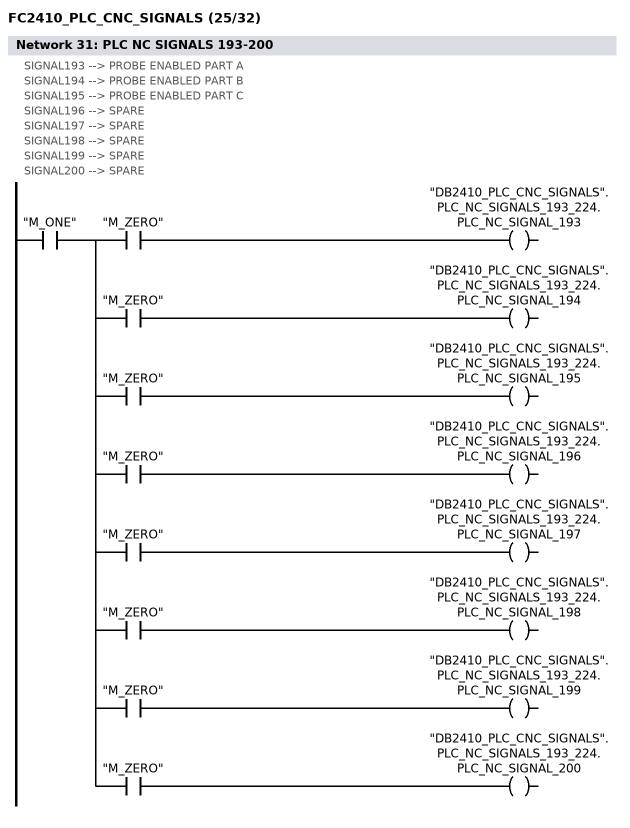
   RUNG wire#powerrail
      Contact( "M_ONE" )
      wire#w1
      Contact( "M_ZERO" )
      Coil( "DB2410_PLC_CNC_SIGNALS".PLC_NC_SIGNALS_193_224.PLC_NC_SIGNAL_193 )
   END_RUNG
   RUNG wire#w1
      Contact( "M_ZERO" )
      Coil( "DB2410_PLC_CNC_SIGNALS".PLC_NC_SIGNALS_193_224.PLC_NC_SIGNAL_194 )
   END_RUNG
   RUNG wire#w1
      Contact( "M_ZERO" )
      Coil( "DB2410_PLC_CNC_SIGNALS".PLC_NC_SIGNALS_193_224.PLC_NC_SIGNAL_195 )
   END_RUNG
   RUNG wire#w1
      Contact( "M_ZERO" )
      Coil( "DB2410_PLC_CNC_SIGNALS".PLC_NC_SIGNALS_193_224.PLC_NC_SIGNAL_196 )
   END_RUNG
   RUNG wire#w1
      Contact( "M_ZERO" )
      Coil( "DB2410_PLC_CNC_SIGNALS".PLC_NC_SIGNALS_193_224.PLC_NC_SIGNAL_197 )
   END_RUNG
   RUNG wire#w1
      Contact( "M_ZERO" )
      Coil( "DB2410_PLC_CNC_SIGNALS".PLC_NC_SIGNALS_193_224.PLC_NC_SIGNAL_198 )
   END_RUNG
   RUNG wire#w1
      Contact( "M_ZERO" )
      Coil( "DB2410_PLC_CNC_SIGNALS".PLC_NC_SIGNALS_193_224.PLC_NC_SIGNAL_199 )
   END_RUNG
   RUNG wire#w1
      Contact( "M_ZERO" )
      Coil( "DB2410_PLC_CNC_SIGNALS".PLC_NC_SIGNALS_193_224.PLC_NC_SIGNAL_200 )
   END_RUNG
   // the same network as SCL:
   "DB2410_PLC_CNC_SIGNALS".PLC_NC_SIGNALS_193_224.PLC_NC_SIGNAL_193 := "M_ONE" AND "M_ZERO";
   "DB2410_PLC_CNC_SIGNALS".PLC_NC_SIGNALS_193_224.PLC_NC_SIGNAL_194 := "M_ONE" AND "M_ZERO";
   "DB2410_PLC_CNC_SIGNALS".PLC_NC_SIGNALS_193_224.PLC_NC_SIGNAL_195 := "M_ONE" AND "M_ZERO";
   "DB2410_PLC_CNC_SIGNALS".PLC_NC_SIGNALS_193_224.PLC_NC_SIGNAL_196 := "M_ONE" AND "M_ZERO";
   "DB2410_PLC_CNC_SIGNALS".PLC_NC_SIGNALS_193_224.PLC_NC_SIGNAL_197 := "M_ONE" AND "M_ZERO";
   "DB2410_PLC_CNC_SIGNALS".PLC_NC_SIGNALS_193_224.PLC_NC_SIGNAL_198 := "M_ONE" AND "M_ZERO";
   "DB2410_PLC_CNC_SIGNALS".PLC_NC_SIGNALS_193_224.PLC_NC_SIGNAL_199 := "M_ONE" AND "M_ZERO";
   "DB2410_PLC_CNC_SIGNALS".PLC_NC_SIGNALS_193_224.PLC_NC_SIGNAL_200 := "M_ONE" AND "M_ZERO";
END_REGION

REGION Network 32: PLC NC SIGNALS 201-208
   // SIGNAL201 --> SPARE
   // SIGNAL202 --> SPARE
   // SIGNAL203 --> SPARE
   // SIGNAL204 --> SPARE
   // SIGNAL205 --> SPARE
   // SIGNAL206 --> SPARE
   // SIGNAL207 --> SPARE
   // SIGNAL208 --> SPARE
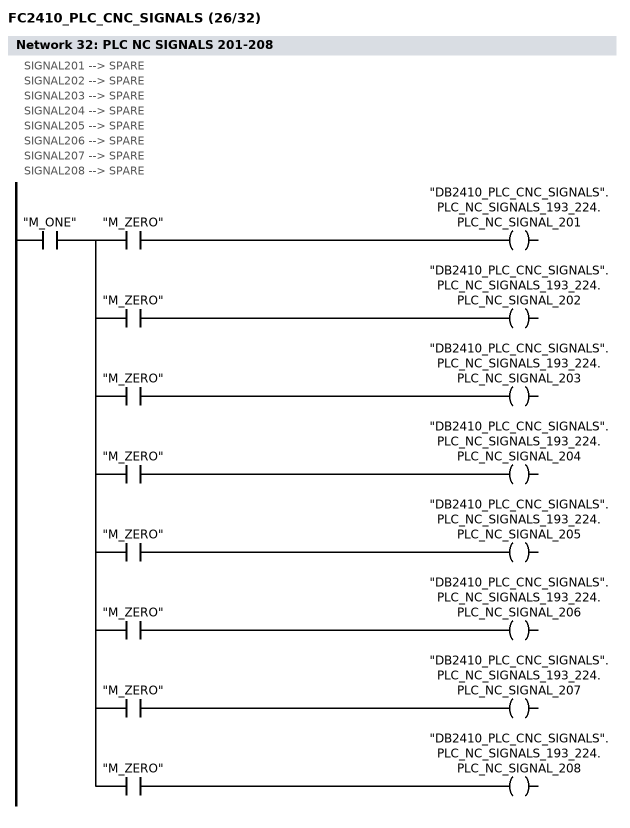
   RUNG wire#powerrail
      Contact( "M_ONE" )
      wire#w1
      Contact( "M_ZERO" )
      Coil( "DB2410_PLC_CNC_SIGNALS".PLC_NC_SIGNALS_193_224.PLC_NC_SIGNAL_201 )
   END_RUNG
   RUNG wire#w1
      Contact( "M_ZERO" )
      Coil( "DB2410_PLC_CNC_SIGNALS".PLC_NC_SIGNALS_193_224.PLC_NC_SIGNAL_202 )
   END_RUNG
   RUNG wire#w1
      Contact( "M_ZERO" )
      Coil( "DB2410_PLC_CNC_SIGNALS".PLC_NC_SIGNALS_193_224.PLC_NC_SIGNAL_203 )
   END_RUNG
   RUNG wire#w1
      Contact( "M_ZERO" )
      Coil( "DB2410_PLC_CNC_SIGNALS".PLC_NC_SIGNALS_193_224.PLC_NC_SIGNAL_204 )
   END_RUNG
   RUNG wire#w1
      Contact( "M_ZERO" )
      Coil( "DB2410_PLC_CNC_SIGNALS".PLC_NC_SIGNALS_193_224.PLC_NC_SIGNAL_205 )
   END_RUNG
   RUNG wire#w1
      Contact( "M_ZERO" )
      Coil( "DB2410_PLC_CNC_SIGNALS".PLC_NC_SIGNALS_193_224.PLC_NC_SIGNAL_206 )
   END_RUNG
   RUNG wire#w1
      Contact( "M_ZERO" )
      Coil( "DB2410_PLC_CNC_SIGNALS".PLC_NC_SIGNALS_193_224.PLC_NC_SIGNAL_207 )
   END_RUNG
   RUNG wire#w1
      Contact( "M_ZERO" )
      Coil( "DB2410_PLC_CNC_SIGNALS".PLC_NC_SIGNALS_193_224.PLC_NC_SIGNAL_208 )
   END_RUNG
   // the same network as SCL:
   "DB2410_PLC_CNC_SIGNALS".PLC_NC_SIGNALS_193_224.PLC_NC_SIGNAL_201 := "M_ONE" AND "M_ZERO";
   "DB2410_PLC_CNC_SIGNALS".PLC_NC_SIGNALS_193_224.PLC_NC_SIGNAL_202 := "M_ONE" AND "M_ZERO";
   "DB2410_PLC_CNC_SIGNALS".PLC_NC_SIGNALS_193_224.PLC_NC_SIGNAL_203 := "M_ONE" AND "M_ZERO";
   "DB2410_PLC_CNC_SIGNALS".PLC_NC_SIGNALS_193_224.PLC_NC_SIGNAL_204 := "M_ONE" AND "M_ZERO";
   "DB2410_PLC_CNC_SIGNALS".PLC_NC_SIGNALS_193_224.PLC_NC_SIGNAL_205 := "M_ONE" AND "M_ZERO";
   "DB2410_PLC_CNC_SIGNALS".PLC_NC_SIGNALS_193_224.PLC_NC_SIGNAL_206 := "M_ONE" AND "M_ZERO";
   "DB2410_PLC_CNC_SIGNALS".PLC_NC_SIGNALS_193_224.PLC_NC_SIGNAL_207 := "M_ONE" AND "M_ZERO";
   "DB2410_PLC_CNC_SIGNALS".PLC_NC_SIGNALS_193_224.PLC_NC_SIGNAL_208 := "M_ONE" AND "M_ZERO";
END_REGION

REGION Network 33: PLC NC SIGNALS 209-216
   // SIGNAL209 --> SPARE
   // SIGNAL210 --> SPARE
   // SIGNAL211 --> SPARE
   // SIGNAL212 --> SPARE
   // SIGNAL213 --> SPARE
   // SIGNAL214 --> SPARE
   // SIGNAL215 --> SPARE
   // SIGNAL216 --> SPARE
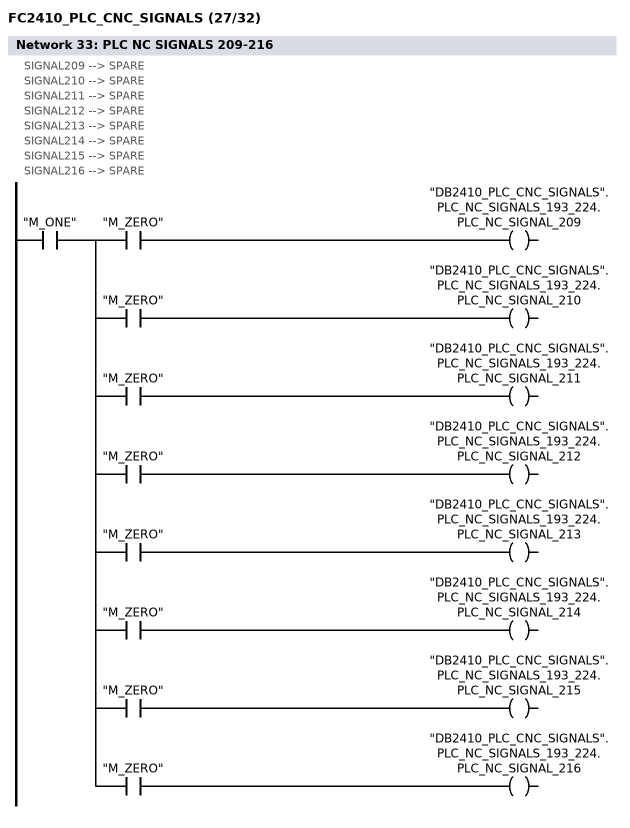
   RUNG wire#powerrail
      Contact( "M_ONE" )
      wire#w1
      Contact( "M_ZERO" )
      Coil( "DB2410_PLC_CNC_SIGNALS".PLC_NC_SIGNALS_193_224.PLC_NC_SIGNAL_209 )
   END_RUNG
   RUNG wire#w1
      Contact( "M_ZERO" )
      Coil( "DB2410_PLC_CNC_SIGNALS".PLC_NC_SIGNALS_193_224.PLC_NC_SIGNAL_210 )
   END_RUNG
   RUNG wire#w1
      Contact( "M_ZERO" )
      Coil( "DB2410_PLC_CNC_SIGNALS".PLC_NC_SIGNALS_193_224.PLC_NC_SIGNAL_211 )
   END_RUNG
   RUNG wire#w1
      Contact( "M_ZERO" )
      Coil( "DB2410_PLC_CNC_SIGNALS".PLC_NC_SIGNALS_193_224.PLC_NC_SIGNAL_212 )
   END_RUNG
   RUNG wire#w1
      Contact( "M_ZERO" )
      Coil( "DB2410_PLC_CNC_SIGNALS".PLC_NC_SIGNALS_193_224.PLC_NC_SIGNAL_213 )
   END_RUNG
   RUNG wire#w1
      Contact( "M_ZERO" )
      Coil( "DB2410_PLC_CNC_SIGNALS".PLC_NC_SIGNALS_193_224.PLC_NC_SIGNAL_214 )
   END_RUNG
   RUNG wire#w1
      Contact( "M_ZERO" )
      Coil( "DB2410_PLC_CNC_SIGNALS".PLC_NC_SIGNALS_193_224.PLC_NC_SIGNAL_215 )
   END_RUNG
   RUNG wire#w1
      Contact( "M_ZERO" )
      Coil( "DB2410_PLC_CNC_SIGNALS".PLC_NC_SIGNALS_193_224.PLC_NC_SIGNAL_216 )
   END_RUNG
   // the same network as SCL:
   "DB2410_PLC_CNC_SIGNALS".PLC_NC_SIGNALS_193_224.PLC_NC_SIGNAL_209 := "M_ONE" AND "M_ZERO";
   "DB2410_PLC_CNC_SIGNALS".PLC_NC_SIGNALS_193_224.PLC_NC_SIGNAL_210 := "M_ONE" AND "M_ZERO";
   "DB2410_PLC_CNC_SIGNALS".PLC_NC_SIGNALS_193_224.PLC_NC_SIGNAL_211 := "M_ONE" AND "M_ZERO";
   "DB2410_PLC_CNC_SIGNALS".PLC_NC_SIGNALS_193_224.PLC_NC_SIGNAL_212 := "M_ONE" AND "M_ZERO";
   "DB2410_PLC_CNC_SIGNALS".PLC_NC_SIGNALS_193_224.PLC_NC_SIGNAL_213 := "M_ONE" AND "M_ZERO";
   "DB2410_PLC_CNC_SIGNALS".PLC_NC_SIGNALS_193_224.PLC_NC_SIGNAL_214 := "M_ONE" AND "M_ZERO";
   "DB2410_PLC_CNC_SIGNALS".PLC_NC_SIGNALS_193_224.PLC_NC_SIGNAL_215 := "M_ONE" AND "M_ZERO";
   "DB2410_PLC_CNC_SIGNALS".PLC_NC_SIGNALS_193_224.PLC_NC_SIGNAL_216 := "M_ONE" AND "M_ZERO";
END_REGION

REGION Network 34: PLC NC SIGNALS 217-224
   // SIGNAL217 --> SPARE
   // SIGNAL218 --> SPARE
   // SIGNAL219 --> SPARE
   // SIGNAL220 --> SPARE
   // SIGNAL221 --> SPARE
   // SIGNAL222 --> SPARE
   // SIGNAL223 --> SPARE
   // SIGNAL224 --> SPARE
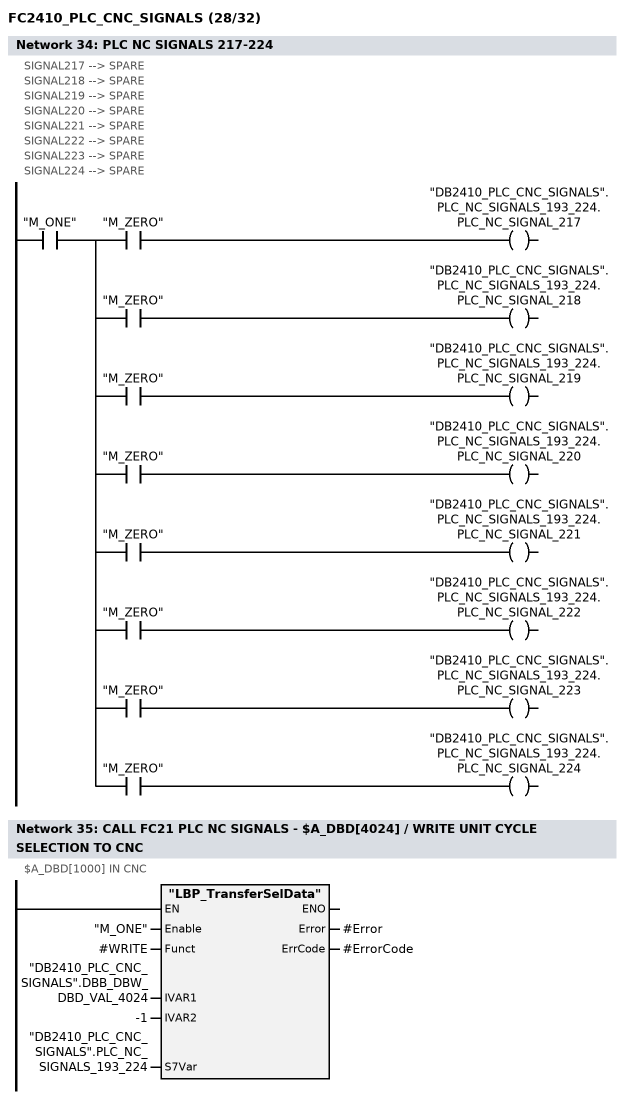
   RUNG wire#powerrail
      Contact( "M_ONE" )
      wire#w1
      Contact( "M_ZERO" )
      Coil( "DB2410_PLC_CNC_SIGNALS".PLC_NC_SIGNALS_193_224.PLC_NC_SIGNAL_217 )
   END_RUNG
   RUNG wire#w1
      Contact( "M_ZERO" )
      Coil( "DB2410_PLC_CNC_SIGNALS".PLC_NC_SIGNALS_193_224.PLC_NC_SIGNAL_218 )
   END_RUNG
   RUNG wire#w1
      Contact( "M_ZERO" )
      Coil( "DB2410_PLC_CNC_SIGNALS".PLC_NC_SIGNALS_193_224.PLC_NC_SIGNAL_219 )
   END_RUNG
   RUNG wire#w1
      Contact( "M_ZERO" )
      Coil( "DB2410_PLC_CNC_SIGNALS".PLC_NC_SIGNALS_193_224.PLC_NC_SIGNAL_220 )
   END_RUNG
   RUNG wire#w1
      Contact( "M_ZERO" )
      Coil( "DB2410_PLC_CNC_SIGNALS".PLC_NC_SIGNALS_193_224.PLC_NC_SIGNAL_221 )
   END_RUNG
   RUNG wire#w1
      Contact( "M_ZERO" )
      Coil( "DB2410_PLC_CNC_SIGNALS".PLC_NC_SIGNALS_193_224.PLC_NC_SIGNAL_222 )
   END_RUNG
   RUNG wire#w1
      Contact( "M_ZERO" )
      Coil( "DB2410_PLC_CNC_SIGNALS".PLC_NC_SIGNALS_193_224.PLC_NC_SIGNAL_223 )
   END_RUNG
   RUNG wire#w1
      Contact( "M_ZERO" )
      Coil( "DB2410_PLC_CNC_SIGNALS".PLC_NC_SIGNALS_193_224.PLC_NC_SIGNAL_224 )
   END_RUNG
   // the same network as SCL:
   "DB2410_PLC_CNC_SIGNALS".PLC_NC_SIGNALS_193_224.PLC_NC_SIGNAL_217 := "M_ONE" AND "M_ZERO";
   "DB2410_PLC_CNC_SIGNALS".PLC_NC_SIGNALS_193_224.PLC_NC_SIGNAL_218 := "M_ONE" AND "M_ZERO";
   "DB2410_PLC_CNC_SIGNALS".PLC_NC_SIGNALS_193_224.PLC_NC_SIGNAL_219 := "M_ONE" AND "M_ZERO";
   "DB2410_PLC_CNC_SIGNALS".PLC_NC_SIGNALS_193_224.PLC_NC_SIGNAL_220 := "M_ONE" AND "M_ZERO";
   "DB2410_PLC_CNC_SIGNALS".PLC_NC_SIGNALS_193_224.PLC_NC_SIGNAL_221 := "M_ONE" AND "M_ZERO";
   "DB2410_PLC_CNC_SIGNALS".PLC_NC_SIGNALS_193_224.PLC_NC_SIGNAL_222 := "M_ONE" AND "M_ZERO";
   "DB2410_PLC_CNC_SIGNALS".PLC_NC_SIGNALS_193_224.PLC_NC_SIGNAL_223 := "M_ONE" AND "M_ZERO";
   "DB2410_PLC_CNC_SIGNALS".PLC_NC_SIGNALS_193_224.PLC_NC_SIGNAL_224 := "M_ONE" AND "M_ZERO";
END_REGION

REGION Network 35: CALL FC21 PLC NC SIGNALS - $A_DBD[4024] / WRITE UNIT CYCLE SELECTION TO CNC
   // $A_DBD[1000] IN CNC
   RUNG wire#powerrail
      "LBP_TransferSelData"(Enable := "M_ONE", Funct := #WRITE, IVAR1 := "DB2410_PLC_CNC_SIGNALS".DBB_DBW_DBD_VAL_4024, IVAR2 := -1, S7Var := "DB2410_PLC_CNC_SIGNALS".PLC_NC_SIGNALS_193_224, Error => #Error, ErrCode => #ErrorCode)
   END_RUNG
   // the same network as SCL:
   "LBP_TransferSelData"(Enable := "M_ONE",
                         Funct := #WRITE,
                         IVAR1 := "DB2410_PLC_CNC_SIGNALS".DBB_DBW_DBD_VAL_4024,
                         IVAR2 := -1,
                         S7Var := "DB2410_PLC_CNC_SIGNALS".PLC_NC_SIGNALS_193_224,
                         Error => #Error,
                         ErrCode => #ErrorCode);
END_REGION

REGION Network 36: PLC NC SIGNALS 225-232
   // SIGNAL225 --> SPARE
   // SIGNAL226 --> SPARE
   // SIGNAL227 --> SPARE
   // SIGNAL228 --> SPARE
   // SIGNAL229 --> SPARE
   // SIGNAL230 --> SPARE
   // SIGNAL231 --> SPARE
   // SIGNAL232 --> SPARE
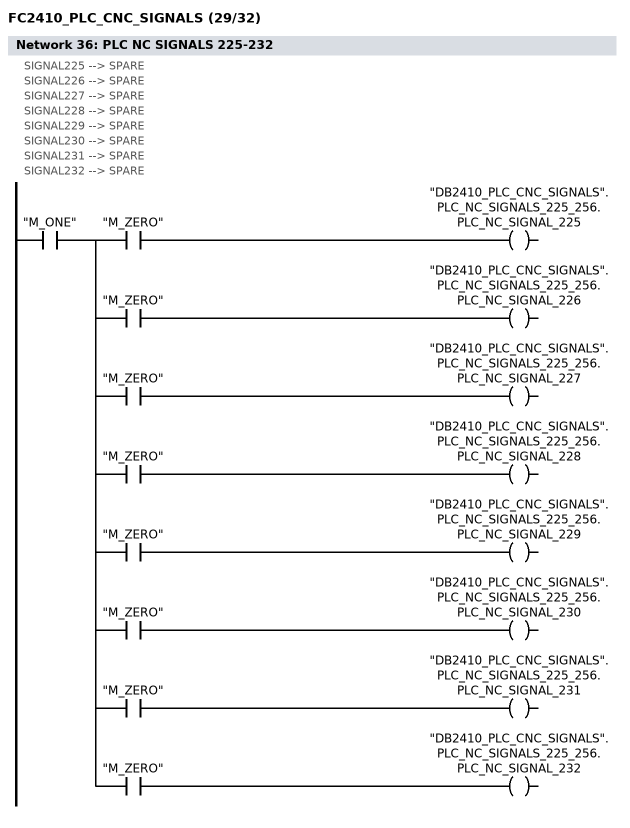
   RUNG wire#powerrail
      Contact( "M_ONE" )
      wire#w1
      Contact( "M_ZERO" )
      Coil( "DB2410_PLC_CNC_SIGNALS".PLC_NC_SIGNALS_225_256.PLC_NC_SIGNAL_225 )
   END_RUNG
   RUNG wire#w1
      Contact( "M_ZERO" )
      Coil( "DB2410_PLC_CNC_SIGNALS".PLC_NC_SIGNALS_225_256.PLC_NC_SIGNAL_226 )
   END_RUNG
   RUNG wire#w1
      Contact( "M_ZERO" )
      Coil( "DB2410_PLC_CNC_SIGNALS".PLC_NC_SIGNALS_225_256.PLC_NC_SIGNAL_227 )
   END_RUNG
   RUNG wire#w1
      Contact( "M_ZERO" )
      Coil( "DB2410_PLC_CNC_SIGNALS".PLC_NC_SIGNALS_225_256.PLC_NC_SIGNAL_228 )
   END_RUNG
   RUNG wire#w1
      Contact( "M_ZERO" )
      Coil( "DB2410_PLC_CNC_SIGNALS".PLC_NC_SIGNALS_225_256.PLC_NC_SIGNAL_229 )
   END_RUNG
   RUNG wire#w1
      Contact( "M_ZERO" )
      Coil( "DB2410_PLC_CNC_SIGNALS".PLC_NC_SIGNALS_225_256.PLC_NC_SIGNAL_230 )
   END_RUNG
   RUNG wire#w1
      Contact( "M_ZERO" )
      Coil( "DB2410_PLC_CNC_SIGNALS".PLC_NC_SIGNALS_225_256.PLC_NC_SIGNAL_231 )
   END_RUNG
   RUNG wire#w1
      Contact( "M_ZERO" )
      Coil( "DB2410_PLC_CNC_SIGNALS".PLC_NC_SIGNALS_225_256.PLC_NC_SIGNAL_232 )
   END_RUNG
   // the same network as SCL:
   "DB2410_PLC_CNC_SIGNALS".PLC_NC_SIGNALS_225_256.PLC_NC_SIGNAL_225 := "M_ONE" AND "M_ZERO";
   "DB2410_PLC_CNC_SIGNALS".PLC_NC_SIGNALS_225_256.PLC_NC_SIGNAL_226 := "M_ONE" AND "M_ZERO";
   "DB2410_PLC_CNC_SIGNALS".PLC_NC_SIGNALS_225_256.PLC_NC_SIGNAL_227 := "M_ONE" AND "M_ZERO";
   "DB2410_PLC_CNC_SIGNALS".PLC_NC_SIGNALS_225_256.PLC_NC_SIGNAL_228 := "M_ONE" AND "M_ZERO";
   "DB2410_PLC_CNC_SIGNALS".PLC_NC_SIGNALS_225_256.PLC_NC_SIGNAL_229 := "M_ONE" AND "M_ZERO";
   "DB2410_PLC_CNC_SIGNALS".PLC_NC_SIGNALS_225_256.PLC_NC_SIGNAL_230 := "M_ONE" AND "M_ZERO";
   "DB2410_PLC_CNC_SIGNALS".PLC_NC_SIGNALS_225_256.PLC_NC_SIGNAL_231 := "M_ONE" AND "M_ZERO";
   "DB2410_PLC_CNC_SIGNALS".PLC_NC_SIGNALS_225_256.PLC_NC_SIGNAL_232 := "M_ONE" AND "M_ZERO";
END_REGION

REGION Network 37: PLC NC SIGNALS 233-240
   // SIGNAL233 --> SPARE
   // SIGNAL234 --> SPARE
   // SIGNAL235 --> SPARE
   // SIGNAL236 --> SPARE
   // SIGNAL237 --> SPARE
   // SIGNAL238 --> SPARE
   // SIGNAL239 --> SPARE
   // SIGNAL240 --> SPARE
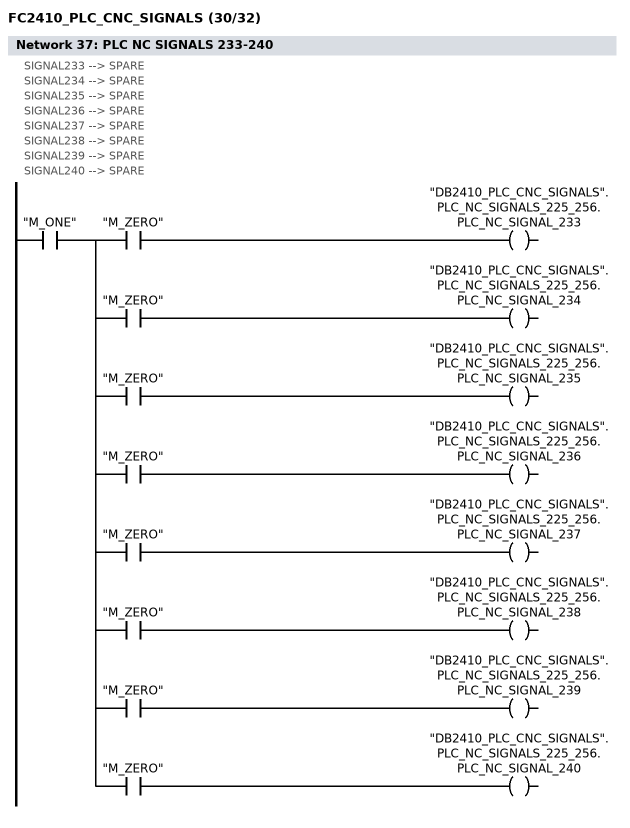
   RUNG wire#powerrail
      Contact( "M_ONE" )
      wire#w1
      Contact( "M_ZERO" )
      Coil( "DB2410_PLC_CNC_SIGNALS".PLC_NC_SIGNALS_225_256.PLC_NC_SIGNAL_233 )
   END_RUNG
   RUNG wire#w1
      Contact( "M_ZERO" )
      Coil( "DB2410_PLC_CNC_SIGNALS".PLC_NC_SIGNALS_225_256.PLC_NC_SIGNAL_234 )
   END_RUNG
   RUNG wire#w1
      Contact( "M_ZERO" )
      Coil( "DB2410_PLC_CNC_SIGNALS".PLC_NC_SIGNALS_225_256.PLC_NC_SIGNAL_235 )
   END_RUNG
   RUNG wire#w1
      Contact( "M_ZERO" )
      Coil( "DB2410_PLC_CNC_SIGNALS".PLC_NC_SIGNALS_225_256.PLC_NC_SIGNAL_236 )
   END_RUNG
   RUNG wire#w1
      Contact( "M_ZERO" )
      Coil( "DB2410_PLC_CNC_SIGNALS".PLC_NC_SIGNALS_225_256.PLC_NC_SIGNAL_237 )
   END_RUNG
   RUNG wire#w1
      Contact( "M_ZERO" )
      Coil( "DB2410_PLC_CNC_SIGNALS".PLC_NC_SIGNALS_225_256.PLC_NC_SIGNAL_238 )
   END_RUNG
   RUNG wire#w1
      Contact( "M_ZERO" )
      Coil( "DB2410_PLC_CNC_SIGNALS".PLC_NC_SIGNALS_225_256.PLC_NC_SIGNAL_239 )
   END_RUNG
   RUNG wire#w1
      Contact( "M_ZERO" )
      Coil( "DB2410_PLC_CNC_SIGNALS".PLC_NC_SIGNALS_225_256.PLC_NC_SIGNAL_240 )
   END_RUNG
   // the same network as SCL:
   "DB2410_PLC_CNC_SIGNALS".PLC_NC_SIGNALS_225_256.PLC_NC_SIGNAL_233 := "M_ONE" AND "M_ZERO";
   "DB2410_PLC_CNC_SIGNALS".PLC_NC_SIGNALS_225_256.PLC_NC_SIGNAL_234 := "M_ONE" AND "M_ZERO";
   "DB2410_PLC_CNC_SIGNALS".PLC_NC_SIGNALS_225_256.PLC_NC_SIGNAL_235 := "M_ONE" AND "M_ZERO";
   "DB2410_PLC_CNC_SIGNALS".PLC_NC_SIGNALS_225_256.PLC_NC_SIGNAL_236 := "M_ONE" AND "M_ZERO";
   "DB2410_PLC_CNC_SIGNALS".PLC_NC_SIGNALS_225_256.PLC_NC_SIGNAL_237 := "M_ONE" AND "M_ZERO";
   "DB2410_PLC_CNC_SIGNALS".PLC_NC_SIGNALS_225_256.PLC_NC_SIGNAL_238 := "M_ONE" AND "M_ZERO";
   "DB2410_PLC_CNC_SIGNALS".PLC_NC_SIGNALS_225_256.PLC_NC_SIGNAL_239 := "M_ONE" AND "M_ZERO";
   "DB2410_PLC_CNC_SIGNALS".PLC_NC_SIGNALS_225_256.PLC_NC_SIGNAL_240 := "M_ONE" AND "M_ZERO";
END_REGION

REGION Network 38: PLC NC SIGNALS 241-248
   // SIGNAL241 --> SPARE
   // SIGNAL242 --> SPARE
   // SIGNAL243 --> SPARE
   // SIGNAL244 --> SPARE
   // SIGNAL245 --> SPARE
   // SIGNAL246 --> SPARE
   // SIGNAL247 --> SPARE
   // SIGNAL248 --> SPARE
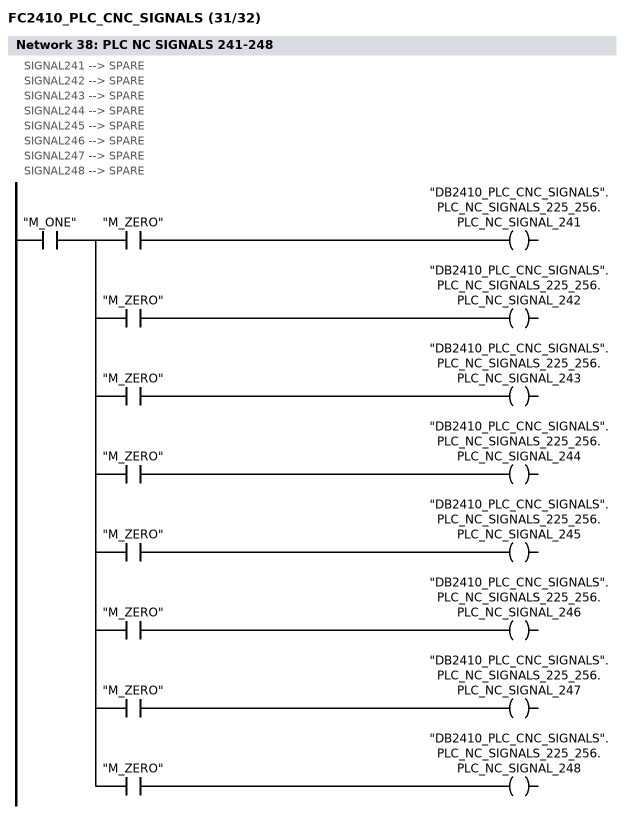
   RUNG wire#powerrail
      Contact( "M_ONE" )
      wire#w1
      Contact( "M_ZERO" )
      Coil( "DB2410_PLC_CNC_SIGNALS".PLC_NC_SIGNALS_225_256.PLC_NC_SIGNAL_241 )
   END_RUNG
   RUNG wire#w1
      Contact( "M_ZERO" )
      Coil( "DB2410_PLC_CNC_SIGNALS".PLC_NC_SIGNALS_225_256.PLC_NC_SIGNAL_242 )
   END_RUNG
   RUNG wire#w1
      Contact( "M_ZERO" )
      Coil( "DB2410_PLC_CNC_SIGNALS".PLC_NC_SIGNALS_225_256.PLC_NC_SIGNAL_243 )
   END_RUNG
   RUNG wire#w1
      Contact( "M_ZERO" )
      Coil( "DB2410_PLC_CNC_SIGNALS".PLC_NC_SIGNALS_225_256.PLC_NC_SIGNAL_244 )
   END_RUNG
   RUNG wire#w1
      Contact( "M_ZERO" )
      Coil( "DB2410_PLC_CNC_SIGNALS".PLC_NC_SIGNALS_225_256.PLC_NC_SIGNAL_245 )
   END_RUNG
   RUNG wire#w1
      Contact( "M_ZERO" )
      Coil( "DB2410_PLC_CNC_SIGNALS".PLC_NC_SIGNALS_225_256.PLC_NC_SIGNAL_246 )
   END_RUNG
   RUNG wire#w1
      Contact( "M_ZERO" )
      Coil( "DB2410_PLC_CNC_SIGNALS".PLC_NC_SIGNALS_225_256.PLC_NC_SIGNAL_247 )
   END_RUNG
   RUNG wire#w1
      Contact( "M_ZERO" )
      Coil( "DB2410_PLC_CNC_SIGNALS".PLC_NC_SIGNALS_225_256.PLC_NC_SIGNAL_248 )
   END_RUNG
   // the same network as SCL:
   "DB2410_PLC_CNC_SIGNALS".PLC_NC_SIGNALS_225_256.PLC_NC_SIGNAL_241 := "M_ONE" AND "M_ZERO";
   "DB2410_PLC_CNC_SIGNALS".PLC_NC_SIGNALS_225_256.PLC_NC_SIGNAL_242 := "M_ONE" AND "M_ZERO";
   "DB2410_PLC_CNC_SIGNALS".PLC_NC_SIGNALS_225_256.PLC_NC_SIGNAL_243 := "M_ONE" AND "M_ZERO";
   "DB2410_PLC_CNC_SIGNALS".PLC_NC_SIGNALS_225_256.PLC_NC_SIGNAL_244 := "M_ONE" AND "M_ZERO";
   "DB2410_PLC_CNC_SIGNALS".PLC_NC_SIGNALS_225_256.PLC_NC_SIGNAL_245 := "M_ONE" AND "M_ZERO";
   "DB2410_PLC_CNC_SIGNALS".PLC_NC_SIGNALS_225_256.PLC_NC_SIGNAL_246 := "M_ONE" AND "M_ZERO";
   "DB2410_PLC_CNC_SIGNALS".PLC_NC_SIGNALS_225_256.PLC_NC_SIGNAL_247 := "M_ONE" AND "M_ZERO";
   "DB2410_PLC_CNC_SIGNALS".PLC_NC_SIGNALS_225_256.PLC_NC_SIGNAL_248 := "M_ONE" AND "M_ZERO";
END_REGION

REGION Network 39: PLC NC SIGNALS 249-256
   // SIGNAL249 --> SPARE
   // SIGNAL250 --> SPARE
   // SIGNAL251 --> SPARE
   // SIGNAL252 --> SPARE
   // SIGNAL253 --> SPARE
   // SIGNAL254 --> SPARE
   // SIGNAL255 --> SPARE
   // SIGNAL256 --> SPARE
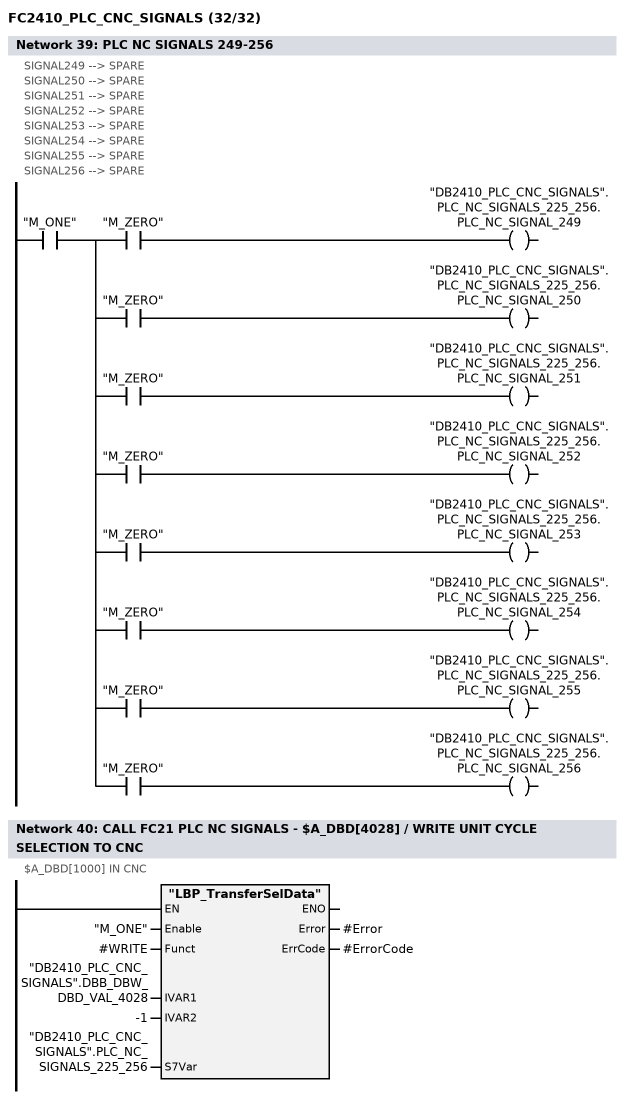
   RUNG wire#powerrail
      Contact( "M_ONE" )
      wire#w1
      Contact( "M_ZERO" )
      Coil( "DB2410_PLC_CNC_SIGNALS".PLC_NC_SIGNALS_225_256.PLC_NC_SIGNAL_249 )
   END_RUNG
   RUNG wire#w1
      Contact( "M_ZERO" )
      Coil( "DB2410_PLC_CNC_SIGNALS".PLC_NC_SIGNALS_225_256.PLC_NC_SIGNAL_250 )
   END_RUNG
   RUNG wire#w1
      Contact( "M_ZERO" )
      Coil( "DB2410_PLC_CNC_SIGNALS".PLC_NC_SIGNALS_225_256.PLC_NC_SIGNAL_251 )
   END_RUNG
   RUNG wire#w1
      Contact( "M_ZERO" )
      Coil( "DB2410_PLC_CNC_SIGNALS".PLC_NC_SIGNALS_225_256.PLC_NC_SIGNAL_252 )
   END_RUNG
   RUNG wire#w1
      Contact( "M_ZERO" )
      Coil( "DB2410_PLC_CNC_SIGNALS".PLC_NC_SIGNALS_225_256.PLC_NC_SIGNAL_253 )
   END_RUNG
   RUNG wire#w1
      Contact( "M_ZERO" )
      Coil( "DB2410_PLC_CNC_SIGNALS".PLC_NC_SIGNALS_225_256.PLC_NC_SIGNAL_254 )
   END_RUNG
   RUNG wire#w1
      Contact( "M_ZERO" )
      Coil( "DB2410_PLC_CNC_SIGNALS".PLC_NC_SIGNALS_225_256.PLC_NC_SIGNAL_255 )
   END_RUNG
   RUNG wire#w1
      Contact( "M_ZERO" )
      Coil( "DB2410_PLC_CNC_SIGNALS".PLC_NC_SIGNALS_225_256.PLC_NC_SIGNAL_256 )
   END_RUNG
   // the same network as SCL:
   "DB2410_PLC_CNC_SIGNALS".PLC_NC_SIGNALS_225_256.PLC_NC_SIGNAL_249 := "M_ONE" AND "M_ZERO";
   "DB2410_PLC_CNC_SIGNALS".PLC_NC_SIGNALS_225_256.PLC_NC_SIGNAL_250 := "M_ONE" AND "M_ZERO";
   "DB2410_PLC_CNC_SIGNALS".PLC_NC_SIGNALS_225_256.PLC_NC_SIGNAL_251 := "M_ONE" AND "M_ZERO";
   "DB2410_PLC_CNC_SIGNALS".PLC_NC_SIGNALS_225_256.PLC_NC_SIGNAL_252 := "M_ONE" AND "M_ZERO";
   "DB2410_PLC_CNC_SIGNALS".PLC_NC_SIGNALS_225_256.PLC_NC_SIGNAL_253 := "M_ONE" AND "M_ZERO";
   "DB2410_PLC_CNC_SIGNALS".PLC_NC_SIGNALS_225_256.PLC_NC_SIGNAL_254 := "M_ONE" AND "M_ZERO";
   "DB2410_PLC_CNC_SIGNALS".PLC_NC_SIGNALS_225_256.PLC_NC_SIGNAL_255 := "M_ONE" AND "M_ZERO";
   "DB2410_PLC_CNC_SIGNALS".PLC_NC_SIGNALS_225_256.PLC_NC_SIGNAL_256 := "M_ONE" AND "M_ZERO";
END_REGION

REGION Network 40: CALL FC21 PLC NC SIGNALS - $A_DBD[4028] / WRITE UNIT CYCLE SELECTION TO CNC
   // $A_DBD[1000] IN CNC
   RUNG wire#powerrail
      "LBP_TransferSelData"(Enable := "M_ONE", Funct := #WRITE, IVAR1 := "DB2410_PLC_CNC_SIGNALS".DBB_DBW_DBD_VAL_4028, IVAR2 := -1, S7Var := "DB2410_PLC_CNC_SIGNALS".PLC_NC_SIGNALS_225_256, Error => #Error, ErrCode => #ErrorCode)
   END_RUNG
   // the same network as SCL:
   "LBP_TransferSelData"(Enable := "M_ONE",
                         Funct := #WRITE,
                         IVAR1 := "DB2410_PLC_CNC_SIGNALS".DBB_DBW_DBD_VAL_4028,
                         IVAR2 := -1,
                         S7Var := "DB2410_PLC_CNC_SIGNALS".PLC_NC_SIGNALS_225_256,
                         Error => #Error,
                         ErrCode => #ErrorCode);
END_REGION
END_FUNCTION
